{attribute 'GeneratedUsingTerminal: EL4732-0001-0000'}
{attribute addProperty BoxType "EL4732-0001-0000"}
{attribute addProperty Id "EtcSlaveTerminalBaseCycle_CounterAT %Q*Cycle_Counter_2C2338042Sample_0AT %Q*Sample_B442BB654WcStateAT %I*WcState_0B2B16F91InfoDataAT %I*InfoData_A7436BC610"}
{attribute addProperty CRC "3315806851"}
{attribute addProperty Size "17"}
TYPE EL4732_C5A33283 EXTENDS EtcSlaveTerminalBase :
STRUCT
	{attribute addProperty Name "Cycle_Counter"}
	Cycle_Counter : Cycle_Counter_2C233804;
	{attribute addProperty Name "Sample_0"}
	Sample_0 : Sample_B442BB65;
	{attribute addProperty Name "WcState"}
	WcState : WcState_0B2B16F9;
	{attribute addProperty Name "InfoData"}
	InfoData : InfoData_A7436BC6;
END_STRUCT
END_TYPE

(* stored: Version 1.2.0.0, ProductVersion 3.1.4024.9
   DUT EL4732_C5A33283: Id {5524ef6d-50fe-47a0-92e1-efd564fd1851} *)
